PROGRAM MAIN
VAR
	
	fbCrossing1 : FB_Crossing;
	(*
	bBool AT%I* : BOOL;
	bBool2 AT%Q* : BOOL;
	nInt1 AT%I* : INT;
	nInt12 AT%Q* : INT;
	nInt13 AT%Q* : INT;
	rTrig : R_TRIG;
	
*)
	
	

END_VAR



fbCrossing1();
(*
rTrig(CLK := bBool);
IF rTrig.Q THEN
	bBool2 := NOT bBool2;
END_IF
*)

END_PROGRAM

(* stored: Version 1.1.0.1, ProductVersion 3.1.4024.0
   POU MAIN: Id {deac02e8-b4b0-4c8f-8c97-6d4c3d73d9f1}, SpecialFunc None *)
